{attribute 'qualified_only'}
VAR_GLOBAL
	icounter : INT;
END_VAR

(* stored: Version 1.1.0.1, ProductVersion 3.1.4024.12
   GVL G_EndMatch: Id {d46e19f3-176b-46ec-a88e-b35d8148b239} *)
